(* CODESYS project MyCustomLibraryPlcProject.library
   Company: My Company
   DefaultNamespace: MyCustomLibrary
   Title: My Custom Library
   Placeholder: MyCustomLibrary
   Author: Your Name
   Version: 1.2.3

Project tree, tasks and I/O mapping:
  libraries: Tc2_System, * (Beckhoff Automation GmbH)
  MyFunctions/
    function MyFunction [ST]
*)

// MyFunctions/MyFunction
FUNCTION MyFunction : T_MAXSTRING
VAR_INPUT
END_VAR
VAR
END_VAR

MyFunction := 'Hello World';

END_FUNCTION
